FUNCTION_BLOCK FB_AxisWithRefSwitch
VAR_INPUT
END_VAR
VAR_OUTPUT
END_VAR
VAR
	prox AT %I* : BOOL;
END_VAR

PROPERTY HomingSensor : BOOL
GET
HomingSensor := prox;
END_GET
END_PROPERTY

END_FUNCTION_BLOCK

(* stored: Version 1.1.0.1, ProductVersion 3.1.4022.18
   POU FB_AxisWithRefSwitch: Id {873109b6-fdee-4331-b6d5-72f8c80c8d32}, SpecialFunc None
   Property HomingSensor: Id {6ab18b84-3041-4610-a46a-ae3856c5c165}
   Get Get: Id {a15d6c32-be12-4f43-9206-cbb7edca1e86} *)
